FUNCTION fcComparePos : BOOL
VAR_INPUT
	CurrPos		:REAL;
	TargetPos	:REAL;
	Tolerance	:REAL;
END_VAR
VAR
END_VAR

IF CurrPos >= 	(TargetPos	-	Tolerance) AND
	CurrPos <= 	(TargetPos	+	Tolerance) THEN
	fcComparePos := TRUE;
ELSE
	fcComparePos := FALSE;
END_IF

END_FUNCTION

(* stored: Version 1.1.0.1, ProductVersion 3.1.4018.2
   POU fcComparePos: Id {d55c393c-b60e-4502-8e43-47725b607f98}, SpecialFunc None *)
